FUNCTION_BLOCK FB_Ejector
VAR_INPUT
END_VAR
VAR_OUTPUT
END_VAR
VAR	
	axis					: FB_Axis;
	zSlide					: FB_Actuator;	
	_Vacuum AT %Q*			: BOOL;
	_VacuumSensor AT %I*	: BOOL;
	_BlowOff AT %Q*			: BOOL;
	_hmiParameters			: ST_EjectorParameters;
	_parameters				: ST_EjectorParameters;
	
	fbMessageChange			: FB_TcMessage;
	fbMessageLoaded			: FB_TcMessage;
	
END_VAR

METHOD Abort : BOOL
VAR_INPUT
END_VAR
BlowOff := FALSE;
PickUpVacuum := FALSE;
zSlide.Neutral();
axis.Disable();
EjectSamplePass(Execute := FALSE);
EjectSampleFail(Execute := FALSE);
Reset(Execute := FALSE);
END_METHOD

PROPERTY BlowOff : BOOL
GET
BlowOff := _BlowOff;
END_GET
SET
_BlowOff := BlowOff;
END_SET
END_PROPERTY

PROPERTY EjectAxisFailPosition : LREAL
GET
EjectAxisFailPosition := _parameters.ejectPositionFail;
END_GET
SET
fbMessageChange.ipArguments.Clear().AddString('EjectAxisFailPosition').AddLReal(_parameters.ejectPositionFail).AddLReal(EjectAxisFailPosition);
fbMessageChange.Send(0);
_parameters.ejectPositionFail := EjectAxisFailPosition;
END_SET
END_PROPERTY

PROPERTY EjectAxisHomePosition : LREAL
GET
EjectAxisHomePosition := _parameters.ejectPositionHome;
END_GET
SET
fbMessageChange.ipArguments.Clear().AddString('EjectAxisHomePosition').AddLReal(_parameters.ejectPositionHome).AddLReal(EjectAxisHomePosition);
fbMessageChange.Send(0);
_parameters.ejectPositionHome := EjectAxisHomePosition;
END_SET
END_PROPERTY

PROPERTY EjectAxisPassPosition : LREAL
GET
EjectAxisPassPosition := _parameters.ejectPositionPass;
END_GET
SET
fbMessageChange.ipArguments.Clear().AddString('EjectAxisPassPosition').AddLReal(_parameters.ejectPositionPass).AddLReal(EjectAxisPassPosition);
fbMessageChange.Send(0);
_parameters.ejectPositionPass := EjectAxisPassPosition;
END_SET
END_PROPERTY

PROPERTY EjectAxisVelocity : LREAL
GET
EjectAxisVelocity := _parameters.ejectVelocity;
END_GET
SET
fbMessageChange.ipArguments.Clear().AddString('EjectAxisVelocity').AddLReal(_parameters.ejectVelocity).AddLReal(EjectAxisVelocity);
fbMessageChange.Send(0);
_parameters.ejectVelocity := EjectAxisVelocity;
END_SET
END_PROPERTY

METHOD EjectSampleFail : INT
VAR_INPUT
	Execute	: BOOL;
END_VAR
VAR_INST
	rTrig	: R_TRIG;
	nIndex	: INT;
	TON		: TON;
	Message	: STRING(255);
END_VAR
VAR
	
END_VAR
EjectSampleFail := 0;
rTrig(CLK := Execute);
IF rTrig.Q THEN
	axis.AbsMove(Execute := FALSE, Position := 0, Velocity := 0);
	nIndex := 10;
END_IF

IF NOT Execute THEN
	nIndex := 0;
END_IF

CASE nIndex OF
	10: // verify that we are retracted in x
		Message := 'Moving to pick up location';
		IF axis.AbsMove(Execute := TRUE, Position := _parameters.ejectPositionHome, Velocity := _parameters.ejectVelocity) THEN
			axis.AbsMove(Execute := FALSE, Position := 0, Velocity := 0);
			nIndex := 20;
		END_IF
		IF axis.Error THEN
			Message := 'Error moving to pick up location';
			axis.AbsMove(Execute := FALSE, Position := 0, Velocity := 0);
			nIndex := 911;
		END_IF
	20: // extend z axis turn on pick up vacuum
		Message := 'Extending z actuator';
		_Vacuum := TRUE;
		IF zSlide.Extend() = 1 THEN
			nIndex := 30;	
		ELSIF zSlide.Extend() = -1 THEN
			Message := 'Error extending z actuator';
			nIndex := 911;
		END_IF
	30: // wait a second
		TON.IN := TRUE;
		TON.PT := T#750MS;
		IF TON.Q THEN
			TON.IN := FALSE;
			nIndex := 40;
		END_IF
		TON();
	40: // retract z axis
		Message := 'Retract z actuator';
		IF zSlide.Retract() = 1 THEN
			nIndex := 50;
		ELSIF zSlide.Retract() = -1 THEN
			Message := 'Error retracting z actuaor';
			nIndex := 911;
		END_IF
	50: // extend the x axis; turn on the blowoff air
		Message := 'Moving to eject reject position';
		IF axis.AbsMove(Execute := TRUE, Position := _parameters.ejectPositionFail, Velocity := _parameters.ejectVelocity) THEN
			axis.AbsMove(Execute := FALSE, Position := 0, Velocity := 0);
			nIndex := 60;
		END_IF
		IF axis.Error THEN
			Message := 'Error moving to reject position';
			nIndex := 911;
			axis.AbsMove(Execute := FALSE, Position := 0, Velocity := 0);
		END_IF
	60: // turn off the blow off	
		_Vacuum := FALSE;	
		IF zSlide.Extend() = 1 THEN
			_BlowOff := TRUE;
		END_IF
		TON.IN := _BlowOff;
		TON.PT := T#500MS;
		IF TON.Q THEN
			_BlowOff := FALSE;		
			TON.IN := FALSE;
			nIndex := 70;
		END_IF
		TON();
	70: // retract the x axis
		Message := 'Moving back to pick up position.';
		zSlide.Retract();
		IF axis.AbsMove(Execute := TRUE, Position := _parameters.ejectPositionHome, Velocity := _parameters.ejectVelocity) THEN
			axis.AbsMove(Execute := FALSE, Position := 0, Velocity := 0);
			nIndex := 80;
		END_IF
		IF axis.Error THEN
			Message := 'Error moving back to pick up position';
			axis.AbsMove(Execute := FALSE, Position := 0, Velocity := 0);
			nIndex := 911;
		END_IF
	80: // done state
		EjectSampleFail := 1;		
END_CASE
END_METHOD

METHOD EjectSamplePass : INT
VAR_INPUT
	Execute	: BOOL;
END_VAR
VAR_INST
	rTrig	: R_TRIG;
	nIndex	: INT;
	TON		: TON;
	Message	: STRING;
END_VAR
EjectSamplePass := 0;
rTrig(CLK := Execute);
IF rTrig.Q THEN
	axis.AbsMove(Execute := FALSE, Position := 0, Velocity := 0);
	nIndex := 10;
END_IF

IF NOT Execute THEN
	nIndex := 0;
END_IF

CASE nIndex OF
	10: // verify that we are retracted in x
		Message := 'Moving to pick up location';
		IF axis.AbsMove(Execute := TRUE, Position := _parameters.ejectPositionHome, Velocity := _parameters.ejectVelocity) THEN
			axis.AbsMove(Execute := FALSE, Position := 0, Velocity := 0);
			nIndex := 20;
		END_IF
		IF axis.Error THEN
			Message := 'Error moving to pick up location';
			axis.AbsMove(Execute := FALSE, Position := 0, Velocity := 0);
			nIndex := 911;
		END_IF
	20: // extend z axis turn on pick up vacuum
		Message := 'Extending z actuator';
		_Vacuum := TRUE;
		IF zSlide.Extend() = 1 THEN
			nIndex := 30;
		ELSIF zSlide.Extend() = -1 THEN
			Message := 'Error extending z actuator';
			nIndex := 911;
		END_IF
	30: // wait a second
		TON.IN := TRUE;
		TON.PT := T#750MS;
		IF TON.Q THEN
			TON.IN := FALSE;
			nIndex := 40;
		END_IF
		TON();
	40: // retract z axis
		Message := 'Retract z actuator';
		IF zSlide.Retract() = 1 THEN
			nIndex := 50;
		ELSIF zSlide.Retract() = -1 THEN
			Message := 'Error retracting z actuaor';
			nIndex := 911;
		END_IF		
	50: // extend the x axis; turn on the blowoff air
		Message := 'Moving to eject pass position';
		IF axis.AbsMove(Execute := TRUE, Position := _parameters.ejectPositionPass, Velocity := _parameters.ejectVelocity) THEN
			axis.AbsMove(Execute := FALSE, Position := 0, Velocity := 0);
			nIndex := 60;
		END_IF
		IF axis.Error THEN
			Message := 'Error moving to pass position';
			nIndex := 911;
			axis.AbsMove(Execute := FALSE, Position := 0, Velocity := 0);
		END_IF
	60: // turn off the blow off		
		_Vacuum := FALSE;
		IF zSlide.Extend() = 1 THEN
			_BlowOff := TRUE;	
		END_IF
		TON.IN := _BlowOff;
		TON.PT := T#500MS;
		IF TON.Q THEN
			_BlowOff := FALSE;		
			TON.IN := FALSE;
			nIndex := 70;
		END_IF
		TON();
	70: // retract the x axis
		Message := 'Moving back to pick up position.';
		zSlide.Retract();
		IF axis.AbsMove(Execute := TRUE, Position := _parameters.ejectPositionHome, Velocity := _parameters.ejectVelocity) THEN
			axis.AbsMove(Execute := FALSE, Position := 0, Velocity := 0);
			nIndex := 80;
		END_IF
		IF axis.Error THEN
			Message := 'Error moving back to pick up position';
			axis.AbsMove(Execute := FALSE, Position := 0, Velocity := 0);
			nIndex := 911;
		END_IF
	80: // done state
		EjectSamplePass := 1;		
END_CASE
END_METHOD

METHOD FB_init : BOOL
VAR_INPUT
	bInitRetains : BOOL; // if TRUE, the retain variables are initialized (warm start / cold start)
	bInCopyCode : BOOL;  // if TRUE, the instance afterwards gets moved into the copy code (online change)
END_VAR
IF NOT fbMessageChange.EqualsToEventEntryEx(stOther := TC_EVENTS.SlitterEvents.ParameterChange) THEN
	fbMessageChange.CreateEx(TC_EVENTS.SlitterEvents.ParameterChange, 0);
	fbMessageChange.ipArguments.Clear();
END_IF

IF NOT fbMessageLoaded.EqualsToEventEntryEx(stOther := TC_EVENTS.SlitterEvents.ParametersLoadedFromFile) THEN
	fbMessageLoaded.CreateEx(TC_EVENTS.SlitterEvents.ParametersLoadedFromFile, 0);
	fbMessageLoaded.ipArguments.Clear().AddString('Ejector');
END_IF
END_METHOD

PROPERTY IsEjectZExtend : BOOL
GET
IsEjectZExtend := zSlide.IsExtended;
END_GET
END_PROPERTY

PROPERTY IsEjectZRetract : BOOL
GET
IsEjectZRetract := zSlide.IsRetracted;
END_GET
END_PROPERTY

METHOD MonitorParameters : BOOL
VAR_INPUT
END_VAR
IF _hmiParameters.ejectPositionFail <> EjectAxisFailPosition THEN
	EjectAxisFailPosition := _hmiParameters.ejectPositionFail;
END_IF

IF _hmiParameters.ejectPositionHome <> EjectAxisHomePosition THEN
	EjectAxisHomePosition := _hmiParameters.ejectPositionHome;
END_IF

IF _hmiParameters.ejectPositionPass <> EjectAxisPassPosition THEN
	EjectAxisPassPosition := _hmiParameters.ejectPositionPass;
END_IF

IF _hmiParameters.ejectVelocity <> EjectAxisVelocity THEN
	EjectAxisVelocity := _hmiParameters.ejectVelocity;
END_IF
END_METHOD

PROPERTY Parameters : ST_EjectorParameters
GET
Parameters := _parameters;
END_GET
SET
fbMessageLoaded.Send(0);
_parameters := Parameters;
_hmiParameters := Parameters;
END_SET
END_PROPERTY

PROPERTY PickUpVacuum : BOOL
GET
PickUpVacuum := _Vacuum;
END_GET
SET
_Vacuum := PickUpVacuum;
END_SET
END_PROPERTY

METHOD Reset : INT
VAR_INPUT
	Execute	: BOOL;
END_VAR
VAR_INST
	rTrig	: R_TRIG;
	nIndex	: INT;
END_VAR
Reset := 0;

rTrig(CLK := Execute);
IF rTrig.Q THEN
	nIndex := 5;
	EjectSampleFail(Execute := FALSE);
	EjectSamplePass(Execute := FALSE);
	axis.AbsMove(Execute := FALSE, Position := 0, Velocity := 0);
	axis.Reset(Execute := FALSE);
END_IF

IF NOT Execute THEN
	nIndex := 0;
END_IF

CASE nIndex OF
	5: 
		BlowOff := FALSE;
		PickUpVacuum := FALSE;
		zSlide.Reset();
		nIndex := 7;
	7: // retract the z axis
		IF zSlide.Retract() = 1 THEN
			nIndex := 10;
		ELSIF zSlide.Retract() = -1 THEN
			nIndex := 911;
		END_IF
		
	10: // disable the axis
		IF axis.Disable() THEN
			nIndex := 20;
		END_IF
	20: // check if there's an error
		IF axis.Error THEN
			nIndex := 30;
		ELSE
			nIndex := 40;
		END_IF
	30: // reset the drive
		IF axis.Reset(Execute := TRUE) THEN
			axis.Reset(Execute := FALSE);
			nIndex := 20;
		END_IF
	40: // enable the drive
		IF axis.Enable() THEN
			nIndex := 50;
		END_IF
	50: // move to the home position
		IF axis.AbsMove(Execute := TRUE, Position := _parameters.ejectPositionHome, Velocity := _parameters.ejectVelocity) THEN
			axis.AbsMove(Execute := FALSE, Position := 0, Velocity := 0);
			nIndex := 60;
		END_IF
		IF axis.Error THEN
			axis.AbsMove(Execute := TRUE, Position := 0, Velocity := 0);
			nIndex := 911;
		END_IF
	60: // done state
		Reset := 1;		
END_CASE
END_METHOD

METHOD ReturnToIdle : INT
VAR_INPUT
END_VAR
_BlowOff := FALSE;
_Vacuum := FALSE;
END_METHOD

END_FUNCTION_BLOCK

(* stored: Version 1.1.0.1, ProductVersion 3.1.4024.9
   POU FB_Ejector: Id {1f9be33f-36d7-436d-adb4-b89b9d7ec6b1}, SpecialFunc None
   Folder Parameters: Id {d8236db4-e37f-4aaa-afb3-c2e28b415a1e}
   Method Abort: Id {9572b01f-15bc-4ea1-bd87-e7c073193092}
   Property BlowOff: Id {bcdb309b-0c76-4954-a549-40664876bfa0}
   Get Get: Id {87ad0e65-5a7a-4c26-9b3e-3d446a1ac2a4}
   Set Set: Id {0a1055a0-a4dc-4e83-8004-d273ac59a5c3}
   Property EjectAxisFailPosition: Id {9325a79d-050a-4ee3-95c1-d06afeab19f3}
   Get Get: Id {81a33da6-85d7-4202-aa27-6d8ec71587a3}
   Set Set: Id {e8b5a0d2-0cc9-4f43-84fd-beb5e04cc5ba}
   Property EjectAxisHomePosition: Id {acdc6ecc-3061-46f9-958d-fe9131ba2c08}
   Get Get: Id {71477ea1-c3e0-484c-b168-81b87fa9761b}
   Set Set: Id {683aab1c-e67b-4e32-a315-d2889294019e}
   Property EjectAxisPassPosition: Id {19ccb745-e931-4dd2-820b-fdf62cb1e7a9}
   Get Get: Id {6cdc2d72-59a7-446c-9aa0-9e71687d0340}
   Set Set: Id {e650fcbf-9c9f-4383-9578-faea53e1bbcc}
   Property EjectAxisVelocity: Id {85234462-7143-4ac0-a2b5-d5f36b8d07e1}
   Get Get: Id {62b18701-363a-4825-9964-c7cd4b23af90}
   Set Set: Id {cb95cddd-8e13-410e-8c0b-f4440e6cbd4f}
   Method EjectSampleFail: Id {3386b649-de86-4924-bd99-2e913152797d}
   Method EjectSamplePass: Id {dd291527-01e2-412b-b66a-fae33418561f}
   Method FB_init: Id {f32fceea-bc73-40fb-bc90-438e4ae6be85}
   Property IsEjectZExtend: Id {1698bd36-a543-499d-b2c9-0725b93a2d39}
   Get Get: Id {463c336d-9028-4e0f-8ae6-4134f2f1d0e5}
   Property IsEjectZRetract: Id {7f9eb240-b4ce-4bd4-9eb4-5bc165852090}
   Get Get: Id {d510e139-e5b2-499d-a913-c5e6609488fe}
   Method MonitorParameters: Id {aab7828f-0417-444b-8c6a-60892fc4f927}
   Property Parameters: Id {fc4dadc5-ad24-4a97-909f-63ba7230c355}
   Get Get: Id {1eeaa37d-857a-42d6-b39d-098c89042a03}
   Set Set: Id {7a5569fd-c4f7-42a9-9263-174e89e2ddb1}
   Property PickUpVacuum: Id {a87a7670-cb9b-4ab4-b830-59f50d3ce68a}
   Get Get: Id {830d474f-9794-4994-a741-5c6b2e06c628}
   Set Set: Id {93930817-90b1-4d77-927b-82f2d2a6e082}
   Method Reset: Id {0548ac50-d050-4ffb-ad43-b2cab5872ecf}
   Method ReturnToIdle: Id {b3aadc4f-bec2-4fa1-88df-a59fbe4935ce} *)
